Staubli VAL3: start.pgx

program start()
begin
clearBuffer(sCal)
taskCreateSync "multi", 0.05, bmulti, multi()
movej(jstart,tGripper,mNomSpeed)
waitEndMove()
taskSuspend("multi")
//operation that does not require sending of data can be performed here
taskResume("multi",1)
movej(jend,tGripper,mNomSpeed)
waitEndMove()
taskSuspend("multi")
taskKill("multi")
end
